// TIA Portal V20 export
TYPE "LAxisCtrl_typeJog"
TITLE = LAxisCtrl_typeJog
// Support: tech.team.motioncontrol@siemens.com 
// Fax: +49 (0) 9131/98-1297
   STRUCT
      velocity : LReal := 0.0;   // Velocity for jogging (Value > 0.0: The specified value is used; Value = 0.0: Permitted; Value < 0.0: The absolute value of the specified value is used)
      acceleration : LReal := -1.0;   // Acceleration for jogging (Value > 0.0: The specified value is used; Value = 0.0: Not permitted; Value < 0.0: Use of the default value configured in the technology object)
      deceleration : LReal := -1.0;   // Deceleration for jogging (Value > 0.0: The specified value is used; Value = 0.0: Not permitted; Value < 0.0: Use of the default value configured in the technology object)
      jerk : LReal := -1.0;   // Jerk for jogging (Value > 0.0: Smooth velocity profile, the specified value is used; Value = 0.0: Trapezoid velocity profile; Value < 0.0: Use of the default value configured in the technology object)
      positionControlled : Bool := TRUE;   // TRUE: Position-controlled mode; FALSE: Non position-controlled operation
      increment : LReal := 0.0;   // Increment/distance for incremental jogging
      mode : DInt := 0;   // 0: Continuous jogging; 1: Incremental jogging new increment (starts with new increment); 2: Incremental jogging continue increment (continue the last increment if not completed)
   END_STRUCT;
END_TYPE
